FUNCTION_BLOCK MonostableCylinder EXTENDS BaseCylinder
VAR_INPUT
END_VAR
VAR_OUTPUT
END_VAR
VAR
END_VAR

METHOD METH_Extend : BOOL
DO_Extend := TRUE;
END_METHOD

METHOD METH_Retract : BOOL
DO_Extend := FALSE;
END_METHOD

END_FUNCTION_BLOCK

(* stored: Version 1.1.0.1, ProductVersion 3.1.4024.9
   POU MonostableCylinder: Id {9c1e3fd3-5a04-4daf-9fa2-9336d8715967}, SpecialFunc None
   Method METH_Extend: Id {46ccace6-d4c6-4ac3-b0f9-6fbe94e9c549}
   Method METH_Retract: Id {af911315-9889-44f1-aa20-5d6308646d45} *)
